(* CODESYS project Exemplo.ecp

Project tree, tasks and I/O mapping:
  Controller : 750-8207 PFC200 CS 2ETH RS 3G, WAGO, order no. 0750-8207, version 5.11.1.16
    application Application
      libraries: ; WagoAppEtherNetIP_Adapter, * (WAGO); WagoAppCloud, * (WAGO)
      task PLC_Task (cyclic, interval t#50ms, priority 15) calls PLC_PRG
      program PLC_PRG [ST]
      program prg_Comunicacao_RockWell [ST]
      data type unionBytes
      global variables g
      program prg_Comunicacao_Nuvem [ST]
    Kbus : Kbus, WAGO, version 1.4.0.2
        unmapped channels: K-BUS diagnostics
    MODBUS
      MODBUS : MODBUS, WAGO, order no. n/a, version 1.1.1.15
    Serial
      COM1 : COM1, WAGO, version 0.0.0.19
      Modem : Modem, WAGO, version 0.0.0.19
*)

// Controller/Application/unionBytes
TYPE unionBytes :
UNION
	aBytes		:		ARRAY[0..31] OF BYTE;
	aReal		:		ARRAY[1..(SIZEOF(aBytes)/4)-1] OF REAL;
	aInt		:		ARRAY[1..(SIZEOF(aBytes)/2)-1] OF INT;
	
END_UNION
END_TYPE

// Controller/Application/g
{attribute 'qualified_only'}
VAR_GLOBAL
	//Módulos Comuns
	rAnalogIN	:	REAL;
	bStatusIN	:	BOOL;
	bStatusOut	:	BOOL;
	rTempIN		:	REAL;
	
	//Módulo de Energia
	rTensaoF1	:	REAL;
	rCorrenteF1	:	REAL;
	rPotAtiva	:	REAL;
	rPotReativa	:	REAL;
	rConsumoKwh	:	REAL;
	
END_VAR

// Controller/Application/PLC_PRG
PROGRAM PLC_PRG
VAR
END_VAR

prg_Comunicacao_RockWell();
prg_Comunicacao_Nuvem();

END_PROGRAM

// Controller/Application/prg_Comunicacao_RockWell
PROGRAM prg_Comunicacao_RockWell
VAR
	//Instância do Bloco de comunicação
	oFb_EthernetIP_Adapter: WagoAppEtherNetIP_Adapter.FbEtherNetIP_Adapter;
	
	xOpen	:	BOOL := TRUE;
	
	oStatus: WagoAppEtherNetIP_Adapter.WagoSysErrorBase.FbResult;
	xError: BOOL;
	xIsOpen: BOOL;
	xIsIdle: BOOL;
	xExclusiveOwnerIsConnected : BOOL;
	xListenOnlyIsConnected		:	BOOL;
	xInputsOnlyIsConnected		:	BOOL;
	oDiagnosis					:	WagoAppEtherNetIP_Adapter.typDiagnosis;
	
	aRxBuffer					:	unionBytes;
	aTxBuffer					:	unionBytes;
	
	
END_VAR

oFb_EthernetIP_Adapter(
	xOpen:= xOpen, 
	oStatus=> oStatus, 
	xError=> xError, 
	xIsOpen=> xIsOpen, 
	xIsIdle=> xIsIdle, 
	eFaultReaction:= eFaultReaction.KeepLastValue, 
	eEthernetNIC:= eEthernetNIC.ethX1_X2, 
	xExclusiveOwnerIsConnected=> xExclusiveOwnerIsConnected, 
	xListenOnlyIsConnected=> xListenOnlyIsConnected, 
	xInputsOnlyIsConnected=> xInputsOnlyIsConnected, 
	oDiagnosis=> oDiagnosis, 
	aRxBuffer:= aRxBuffer.aBytes, 
	aTxBuffer:= aTxBuffer.aBytes);
	
	//Variáveis Globais.
	g.rTensaoF1 	:=	aRxBuffer.aReal[1]; // Transferindo Tensão.
	g.rCorrenteF1	:=	aRxBuffer.aReal[2]; // Recebendo Corrente.
	g.rPotAtiva 	:=	aRxBuffer.aReal[3]; // Recebendo Potência Ativa;
	g.rPotReativa	:=	aRxBuffer.aReal[4];	// Recebendo Potência Reativa;
	g.rConsumoKwh	:=	aRxBuffer.aReal[5]; // Recendo Consumo KWH
	g.rTempIN		:=	aRxBuffer.aReal[6]; // Recebendo Tempereatura ºC
	
	g.rAnalogIN		:=	aRxBuffer.aReal[7]; // Recebendo sinal 0 .. 10V;
	g.bStatusIN		:=	aRxBuffer.aBytes[28].0;// Recebendo sinal digital de entrada
	g.bStatusOut	:=	aRxBuffer.aBytes[28].1;// Recebendo sinal digital de saída

END_PROGRAM

// Controller/Application/prg_Comunicacao_Nuvem
PROGRAM prg_Comunicacao_Nuvem
VAR
	fbCollection 	: 	WagoAppCloud.FbCollectionLogger;
	fbMyCollections	:	WagoAppCloud.typCollection;
	variaveis		:	ARRAY[1..9] OF WagoAppCloud.typVariableDescription;
	oStatus			:	WagoSysErrorBase.FbResult;
END_VAR

VAR RETAIN
	tSampleTime1 : 	TIME := T#2500MS;
	tPublishTime1:	TIME := T#5S;
END_VAR


fbMyCollections.dwCollectionId := 1;
fbMyCollections.sName := 'Variáveis do Compact L33ER';
fbMyCollections.pSampleInterval := ADR(tSampleTime1);
fbMyCollections.pPublishInterval := ADR(tPublishTime1);
fbMyCollections.pVariableDescriptions := ADR(variaveis);
fbMyCollections.dwVariablesCount := 9;


variaveis[1].sTag := 'TensãoF1';
variaveis[1].pAddress := ADR(g.rTensaoF1);
variaveis[1].eValueType := WagoAppCloud.VVT_REAL;
variaveis[1].dwTypeId := 1;
variaveis[1].sUnit := 'V';

variaveis[2].sTag := 'CorrenteF1';
variaveis[2].pAddress := ADR(g.rCorrenteF1);
variaveis[2].eValueType := WagoAppCloud.VVT_REAL;
variaveis[2].dwTypeId := 2;
variaveis[2].sUnit := 'A';

variaveis[3].sTag := 'PotAtivaF1';
variaveis[3].pAddress := ADR(g.rPotAtiva);
variaveis[3].eValueType := WagoAppCloud.VVT_REAL;
variaveis[3].dwTypeId := 3;
variaveis[3].sUnit := 'W';

variaveis[4].sTag := 'PotReativaF1';
variaveis[4].pAddress := ADR(g.rPotReativa);
variaveis[4].eValueType := WagoAppCloud.VVT_REAL;
variaveis[4].dwTypeId := 4;
variaveis[4].sUnit := 'VAr';

variaveis[5].sTag := 'Consumo Total';
variaveis[5].pAddress := ADR(g.rConsumoKwh);
variaveis[5].eValueType := WagoAppCloud.VVT_REAL;
variaveis[5].dwTypeId := 5;
variaveis[5].sUnit := 'Wh';

variaveis[6].sTag := 'Temperatura';
variaveis[6].pAddress := ADR(g.rTempIN);
variaveis[6].eValueType := WagoAppCloud.VVT_REAL;
variaveis[6].dwTypeId := 6;
variaveis[6].sUnit := 'ºC';

variaveis[7].sTag := 'Entrada Analogica';
variaveis[7].pAddress := ADR(g.rAnalogIN);
variaveis[7].eValueType := WagoAppCloud.VVT_REAL;
variaveis[7].dwTypeId := 7;
variaveis[7].sUnit := 'V';

variaveis[8].sTag := 'Sensor';
variaveis[8].pAddress := ADR(g.bStatusIN);
variaveis[8].eValueType := WagoAppCloud.VVT_BOOL;
variaveis[8].dwTypeId := 8;
variaveis[8].sUnit := 'bit';

variaveis[9].sTag := 'LED';
variaveis[9].pAddress := ADR(g.bStatusOut);
variaveis[9].eValueType := WagoAppCloud.VVT_BOOL;
variaveis[9].dwTypeId := 9;
variaveis[9].sUnit := 'bit';

fbCollection(pCollections:=ADR(fbMyCollections),dwCollectionsCount:=1,oStatus => oStatus);

END_PROGRAM
